Fanuc KAREL source: kb00076.KL

-- PROVISIONAL review KL for V1013-1; original PC SHA256 2b813ac9a9be8e81fe75d51c49ccfeed5b3dbd80cf9d43407e73bb365263a97d
-- Incomplete behavior may be omitted. Consult companion uncertainty JSON. Do not deploy.
PROGRAM KB00076
%NOLOCKGROUP
-- UNRESOLVED_DECL P1 type=000101
-- UNRESOLVED_DECL P2 type=000101
-- UNRESOLVED_DECL P3 type=000101
-- UNRESOLVED_DECL RESULT type=000101
BEGIN
  -- UNRESOLVED_PC offsets 5-56; opcodes 27,22,1C,22,1C,22,1C,76,7E,4A
  -- UNRESOLVED_PC offsets 61-65; opcodes 7F
END KB00076
